Universal Robots URScript: step5d_contact_relief_v1.script

# VERSION: 2026-09-20T1458Z_CONTACT_RELIEF_V1
# ROLE: monitored Base +Z relief only; no XY or attitude transfer
# No force-control restart; host owns fresh Kunwei unloading guard and Stop.
def codex_start_hover_finite_value(value, absolute_limit):
  if value != value:
    return False
  end
  if value > absolute_limit or value < -absolute_limit:
    return False
  end
  return True
end

def codex_start_hover_finite_pose(pose_value):
  local index = 0
  while index < 6:
    if not codex_start_hover_finite_value(pose_value[index], 100.0):
      return False
    end
    index = index + 1
  end
  return True
end

def codex_start_hover_motion_limits_ok():
  local segment_1_accel_m_s2 = 0.060
  local segment_1_speed_m_s = 0.040
  local segment_2_accel_m_s2 = 0.135
  local segment_2_speed_m_s = 0.090
  if segment_1_accel_m_s2 <= 0.0 or segment_1_accel_m_s2 > 0.150000000:
    return False
  end
  if segment_2_accel_m_s2 <= 0.0 or segment_2_accel_m_s2 > 0.150000000:
    return False
  end
  if segment_1_speed_m_s <= 0.0 or segment_1_speed_m_s > 0.100000000:
    return False
  end
  if segment_2_speed_m_s <= 0.0 or segment_2_speed_m_s > 0.100000000:
    return False
  end
  return True
end

def codex_start_hover_target_within_limits(target_pose):
  if not codex_start_hover_finite_pose(target_pose):
    return False
  end
  if target_pose[0] < 0.300000000 or target_pose[0] > 0.700000000:
    return False
  end
  if target_pose[1] < -0.200000000 or target_pose[1] > 0.400000000:
    return False
  end
  if target_pose[2] < 0.025000000 or target_pose[2] > 0.200000000:
    return False
  end
  local rotation_norm_rad = sqrt(target_pose[3] * target_pose[3] + target_pose[4] * target_pose[4] + target_pose[5] * target_pose[5])
  if rotation_norm_rad > 3.200000000:
    return False
  end
  return codex_start_hover_motion_limits_ok()
end

def codex_start_hover_final_stationary_verified(target_pose):
  local actual_pose = get_actual_tcp_pose()
  if not codex_start_hover_finite_pose(actual_pose):
    return False
  end
  local actual_speed = get_actual_tcp_speed()
  local actual_joint_speed = get_actual_joint_speeds()
  local speed_index = 0
  local joint_speed_max_rad_s = 0.0
  while speed_index < 6:
    if not codex_start_hover_finite_value(actual_speed[speed_index], 100.0):
      return False
    end
    if not codex_start_hover_finite_value(actual_joint_speed[speed_index], 100.0):
      return False
    end
    local joint_speed_abs = actual_joint_speed[speed_index]
    if joint_speed_abs < 0.0:
      joint_speed_abs = -joint_speed_abs
    end
    if joint_speed_abs > joint_speed_max_rad_s:
      joint_speed_max_rad_s = joint_speed_abs
    end
    speed_index = speed_index + 1
  end
  local delta_pose = pose_trans(pose_inv(target_pose), actual_pose)
  local position_error_m = sqrt(delta_pose[0] * delta_pose[0] + delta_pose[1] * delta_pose[1] + delta_pose[2] * delta_pose[2])
  local orientation_error_rad = sqrt(delta_pose[3] * delta_pose[3] + delta_pose[4] * delta_pose[4] + delta_pose[5] * delta_pose[5])
  local linear_speed_m_s = sqrt(actual_speed[0] * actual_speed[0] + actual_speed[1] * actual_speed[1] + actual_speed[2] * actual_speed[2])
  local angular_speed_rad_s = sqrt(actual_speed[3] * actual_speed[3] + actual_speed[4] * actual_speed[4] + actual_speed[5] * actual_speed[5])
  if position_error_m != position_error_m or orientation_error_rad != orientation_error_rad:
    return False
  end
  if linear_speed_m_s != linear_speed_m_s or angular_speed_rad_s != angular_speed_rad_s:
    return False
  end
  return position_error_m <= 0.003000000 and orientation_error_rad <= 0.050000000 and linear_speed_m_s <= 0.001000000 and angular_speed_rad_s <= 0.010000000 and joint_speed_max_rad_s <= 0.010000000
end


def step5d_contact_relief_v1():
  local current_pose = get_actual_tcp_pose()
  local target_pose = p[0.487834547, 0.129337053, 0.033, 2.0331342431227566, 2.3949884238824652, -2.2711768777011217e-22]
  if not codex_start_hover_finite_pose(current_pose):
    halt
  end
  local dx = current_pose[0]-target_pose[0]
  local dy = current_pose[1]-target_pose[1]
  local dz = current_pose[2]-target_pose[2]
  local distance = sqrt(dx*dx + dy*dy + dz*dz)
  local turn = pose_trans(pose_inv(target_pose), current_pose)
  local angle = sqrt(turn[3]*turn[3] + turn[4]*turn[4] + turn[5]*turn[5])
  if distance > 0.080 or angle > 0.010 or current_pose[2] < 0.018 or current_pose[2] > 0.034:
    textmsg("contact_relief: initial geometry rejected")
    halt
  end
  if current_pose[2] < 0.033:
    local rise_pose = p[current_pose[0], current_pose[1], 0.033, current_pose[3], current_pose[4], current_pose[5]]
    movel(rise_pose, a=0.005, v=0.0005, r=0.0)
    stopl(0.1)
  end
  sleep(0.20)
  textmsg("contact_relief: vertical stage complete; awaiting host release check")
  halt
end

step5d_contact_relief_v1()
